Fanuc KAREL source: compact_preamble.KL

PROGRAM KT00957
%NOLOCKGROUP
VAR
ENTRY:INTEGER;PNAME : STRING[80];VNAME : STRING[80];STATUS:INTEGER;VALUE:REAL
BEGIN
ENTRY=0
PNAME=''
VNAME='VALUE'
SET_VAR(ENTRY,PNAME,VNAME,VALUE,STATUS)
END KT00957
